// TIA Portal V21 export
DATA_BLOCK "DB607"   // DB607
AUTHOR : PRECISE
FAMILY : PRECISE
// stored: AutoNumber false, InstanceOfName FB607, InstanceOfType FB
"FB607"
   // VAR_INPUT
   //    CipSelected : Bool;
   //    CycleEnable : Bool;
   //    CycleRunning : Bool;
   //    SecPulse : Bool;
   //    AlwaysTrue : Bool;
   //    MixingTimeBaseSel : Bool;
   //    SetTimeMins : Int;
   //    SetTimeSecs : Int;
   //    ActualRepetition : Int;
   // END_VAR
   // VAR_OUTPUT
   //    Started : Bool;
   //    Mixer : Bool;
   //    TimeMinsPv : DInt;
   //    TimeSecsPv : DInt;
   //    StepStatus : String[60];
   //    Print : "MixingPrint";
   // END_VAR
   // VAR_IN_OUT
   //    Over : Bool;
   // END_VAR
   // VAR
   //    RE1 : Bool;
   //    RE2 : Bool;
   //    RE3 : Bool;
   //    MixingTimer { S7_SetPoint := 'True'} : "FB101";
   // END_VAR
BEGIN
END_DATA_BLOCK
